FUNCTION_BLOCK I_GetAttribute (* Command GetAttribute( Part 6 - F.58 ) *)
  (* Standard: ISO 11783-6; Description: Copyright (c) 2022 HR Agrartechnik GmbH This program and the accompanying materials are made available under the terms of the Eclipse Public License 2.0 which is available at https://www.eclipse.org/legal/epl-2.0/ SPDX-License-Identifier: EPL-2.0 see Description Tab *)
  (* Version 1.0, 2022-07-08, Franz Höpfinger, HR Agrartechnik GmbH *)
  PACKAGE isobus::UT::I;
  IMPORT isobus::UT::Q::const::IDs::ID_NULL;
  (* Documentation:
  Command GetAttribute( Part 6 - F.58 )
   This message is available in VT Version 4 and later. This command is used by a Working Set to query the VT for the current state of objects within the VT.
   Valid values for u16ObjId
   The Get Attribute Value command (F.58) is a fixed 8-byte message (Object ID in bytes 2,3, Attribute ID in Byte 4; no Transport Protocol). INIT validates both the object type (iso_has_readable_attribute_id - does this object type have any AID at all, read-only or writable?) and the specific Attribute ID against that type's attribute table (iso_is_readable_attribute), before the command is ever sent - unlike Change Attribute, both read-only and writable AIDs are accepted here. The underlying C implementation itself (cmd_get_attribute_value) performs no type check of its own, only ID_NULL handling; the VT additionally validates the Object ID and the Attribute ID on its side and returns an error response if either is invalid.
   ID_NULL (65535) is not a command target but can be used in INIT to deactivate the FB.
   param[in] {objectID, uint16_t}
   Object ID
   param[in] {attributeID, uint8_t}
   Attribute ID of the object
   Return Values: 
   int16_t
    - VT_E_NO_ERR (0) - OK
   - VT_E_DEACTIVATED (-40) - FB deactivated via ID_NULL on INIT
   - VT_E_INVALID_OBJECT_ID (-132) - Object ID's type has no readable AID at all (iso_has_readable_attribute_id)
   - VT_E_INVALID_ATTRIBUTE_ID (-133) - Attribute ID is not a valid/readable AID for this object type (iso_is_readable_attribute)
   - VT_E_NOT_READY (-131) - Buffered: INIT not yet completed / VT not yet ready
   - VT_E_OVERFLOW (-6) - buffer overflow
   - VT_E_NOACT (-8) - Command not possible in current state
   - VT_E_NO_INSTANCE (-21) - No VT client available
   - VT_E_HANDLE_INVALID (-128) - ErrorCause: invalid Handle
   - VT_E_ISO_INSTANCE_INVALID (-129) - Identifier for instance (connection) invalid
   - VT_E_NOT_ALIVE (-130) - Identifier for instance valid, but VT Dead.
    Instanz-Eindeutigkeit (Instance Uniqueness)
   Dieser Baustein erfordert Instanz-Eindeutigkeit bezüglich des Paares (u16ObjId, u8AID). Es darf im gesamten Programm nur eine Instanz von I_GetAttribute für dasselbe Objekt-Attribut-Paar existieren. u8AID wird bei INIT eingelesen — eine zweite Instanz auf dieselbe Objekt-ID und Attribut-ID wird bei INIT deaktiviert.
  *)
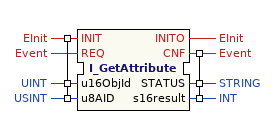
  EVENT_INPUT
    INIT : EInit WITH u16ObjId, u8AID; (* Service Initialization *)
    REQ; (* Service Request *)
  END_EVENT
  EVENT_OUTPUT
    INITO : EInit; (* Initialization Confirm *)
    CNF WITH STATUS, s16result; (* Confirmation of Requested Service *)
  END_EVENT
  VAR_INPUT
    u16ObjId : UINT := ID_NULL; (* Object ID *)
    u8AID : USINT; (* Attribute ID of the object *)
  END_VAR
  VAR_OUTPUT
    STATUS : STRING; (* Service Status *)
    s16result : INT; (* retval see description *)
  END_VAR
END_FUNCTION_BLOCK
